PROGRAM EventGrid
VAR
	fbEventlogger : FB_TcEventLogger;
	fbAlarm: FB_TcAlarm;
	fbMessage: FB_TcMessage;
	bAlarm: BOOL;
	bMessage : BOOL;
	bIsInitalized: BOOL;
	bClearAlarm: BOOL;
	bConfirmAlarm: BOOL;
END_VAR

IF NOT bIsInitalized THEN
	bIsInitalized := TRUE;
	fbMessage.CreateEx(TC_Events.Sinterstar_Mini_EventClass.Sinterstar_Mini_EventClassEvent2, 0);
	fbAlarm.CreateEx(TC_Events.Sinterstar_Mini_EventClass.Sinterstar_Mini_EventClassEvent2, TRUE, 0);
END_IF

IF bMessage THEN
	bMessage := FALSE;
	fbMessage.Send(0);
END_IF

IF bAlarm THEN
	bAlarm := FALSE;
	fbAlarm.Raise(0);
END_IF

IF bClearAlarm THEN
	bClearAlarm := FALSE;
	fbAlarm.Clear(0, FALSE);
END_IF

END_PROGRAM

(* stored: Version 1.1.0.1, ProductVersion 3.1.4024.12
   POU EventGrid: Id {2c02faee-bff7-4e64-a9cf-422fb345f0c4}, SpecialFunc None *)
